# EPICS autosave request: iocBoot/ioc13lab/auto_settings.req
file "scaler_settings.req", P=$(P), S=scaler1
file "scaler_settings.req", P=$(P), S=scaler2
file "scan_settings.req", P=$(P), S=scan1
file "scan_settings.req", P=$(P), S=scan2
file "scan_settings.req", P=$(P), S=scan3
file "scan_settings.req", P=$(P), S=scan4
file "saveData_settings.req", P=$(P)
file "Keithley2kDMM_mf10_settings.req", P=$(P), Dmm=DMM1
file "Keithley2kDMM_mf10_settings.req", P=$(P), Dmm=DMM2
file "Fluke_8842A_settings.req", P=$(P), M=Fluke1
file "Pelco_CM6700_settings.req", P=$(P), R=Pelco1
#file "SR630_settings.req", P=$(P), R=TC1, N=1
#file "SR630_settings.req", P=$(P), R=TC1, N=2
#file "SR630_settings.req", P=$(P), R=TC1, N=3
#file "SR630_settings.req", P=$(P), R=TC1, N=4
#file "SR630_settings.req", P=$(P), R=TC1, N=5
#file "SR630_settings.req", P=$(P), R=TC1, N=6
#file "SR630_settings.req", P=$(P), R=TC1, N=7
#file "SR630_settings.req", P=$(P), R=TC1, N=8
#file "SR630_settings.req", P=$(P), R=TC1, N=9
#file "SR630_settings.req", P=$(P), R=TC1, N=10
#file "SR630_settings.req", P=$(P), R=TC1, N=11
#file "SR630_settings.req", P=$(P), R=TC1, N=12
#file "SR630_settings.req", P=$(P), R=TC1, N=13
#file "SR630_settings.req", P=$(P), R=TC1, N=14
#file "SR630_settings.req", P=$(P), R=TC1, N=15
#file "SR630_settings.req", P=$(P), R=TC1, N=16
file "ccd_settings.req",P=$(P),C=ccd1
file "icb_amp_settings.req", P=$(P), AMP=amp1
file "icb_adc_settings.req", P=$(P), ADC=adc1
file "icb_hvps_settings.req", P=$(P), HVPS=hvps1
file "icb_tca_settings.req", P=$(P), TCA=tca1
file "mca_settings.req", P=$(P), M=aim_adc1
file "mca_settings.req", P=$(P), M=aim_adc2
file "simple_mca_settings.req", P=$(P)quadEM:, M=mca1
file "simple_mca_settings.req", P=$(P)quadEM:, M=mca2
file "simple_mca_settings.req", P=$(P)quadEM:, M=mca3
file "simple_mca_settings.req", P=$(P)quadEM:, M=mca4
file "simple_mca_settings.req", P=$(P)quadEM:, M=mca5
file "simple_mca_settings.req", P=$(P)quadEM:, M=mca6
file "simple_mca_settings.req", P=$(P)quadEM:, M=mca7
file "simple_mca_settings.req", P=$(P)quadEM:, M=mca8
file "simple_mca_settings.req", P=$(P)quadEM:, M=mca9
file "simple_mca_settings.req", P=$(P)quadEM:, M=mca10
file "quadEM_settings.req", P=$(P), EM=EM1
file "pseudoMotor_settings.req", P=$(P), M=pm1
file "pseudoMotor_settings.req", P=$(P), M=pm2
file "CARS_16_motor_settings.req", P=$(P)
$(P)m32.PCOF
$(P)m32.ICOF
$(P)m32.DCOF
